PROGRAM A_2_PRG_MachineCtrl
VAR
/////////////////////////////////////////////////////////////////////////////////////TIMERS & TRIGGERS/////////////////////////////////////////////////////////////////////////////////////

	tonSys_Init					: Tc2_Standard.TON:=(PT:=T#1S);
	tonSys_InitTimeout			: Tc2_Standard.TON:=(PT:=T#20S);					
	tonFirstAutoCycle			: Tc2_Standard.TON:=(PT:=T#500MS);
	
/////////////////////////////////////////////////////////////////////////////////////PROCESS CYCLE/////////////////////////////////////////////////////////////////////////////////////	
	
	eCycleState					: E_ProcessCycle;
	tonCMD_Done					: TON;
	tonResetAllCMD				: TON;
	tonExecute					: TON;
	tonSave_Data				: TON;
	tonWriteToCsv				: TON;
	rNoAutoCycle				: R_TRIG;
	
	bStartProcessCondition		: BOOL;
	bIndexDataHistoryFlag		: BOOL;
	rIndexDataHistoryFlag		: R_TRIG;
	bPASS						: BOOL;
	bFAIL						: BOOL;
	i							: INT;
	

	
END_VAR

/////////////////////////////////////////////////////////////////////////////////////GENERAL/////////////////////////////////////////////////////////////////////////////////////
a_ACT_MachineStatus();
b_ACT_ProcessCycle();

ACTION a_ACT_MachineStatus:
/////////////////////////////////////////////////////////////////////////////////////TIMERS/////////////////////////////////////////////////////////////////////////////////////
tonSys_Init(IN:=stMachineStatus.bInitialising);
tonSys_InitTimeout(IN:=stMachineStatus.bInitialising);


/////////////////////////////////////////////////////////////////////////////////////CONDITIONS/////////////////////////////////////////////////////////////////////////////////////
				IF NOT stMasterCtrl.bNoImmediateFault THEN
					stMachineStatus.eMachineState 		:= E_MachineState.IMMEDIATE_FAULT;
				END_IF
				
				IF stMachineStatus.eMachineState		= E_MachineState.STOPPING OR
				stMachineStatus.eMachineState			= E_MachineState.IMMEDIATE_FAULT OR
				stMachineStatus.eMachineState			= E_MachineState.CYCLE_STOP_FAULT THEN
					
					CMD_Station1.bAbort					:= TRUE;	
					CMD_Station2.bAbort					:= TRUE;	
					CMD_Station3.bAbort					:= TRUE;
				
					CMD_Station1.bEnable				:= FALSE;
					CMD_Station2.bEnable				:= FALSE;
					CMD_Station3.bEnable				:= FALSE;
					
				END_IF
				
				IF 	stButtonsLamps.bResetButtonFallingEdge THEN
					CMD_Station1.bReset					:= TRUE;
					CMD_Station2.bReset					:= TRUE;
					CMD_Station3.bReset					:= TRUE;
				ELSE 
					CMD_Station1.bReset					:= FALSE;
					CMD_Station2.bReset					:= FALSE;
					CMD_Station3.bReset					:= FALSE;
				END_IF		
				
/////////////////////////////////////////////////////////////////////////////////////MACHINE CONTROL/////////////////////////////////////////////////////////////////////////////////////

CASE stMachineStatus.eMachineState OF

E_MachineState.SYSTEM_POWER_UP: 		

				IF tonSystemPowerUP.Q THEN
						stMachineStatus.eMachineState 	:= E_MachineState.IMMEDIATE_STOPPED;//
				END_IF
	
E_MachineState.IMMEDIATE_STOPPED:		

				IF stButtonsLamps.bResetButtonFallingEdge THEN
						stMachineStatus.eMachineState 	:= E_MachineState.SYSTEM_INITIALISING;//
				END_IF	


E_MachineState.SYSTEM_INITIALISING:		
				
				CMD_Station1.bAbort						:= FALSE;	
				CMD_Station2.bAbort						:= FALSE;	
				CMD_Station3.bAbort						:= FALSE;	

				IF tonSys_Init.Q THEN
					CMD_Station1.bEnable				:= TRUE;
					CMD_Station2.bEnable				:= TRUE;
					CMD_Station3.bEnable				:= TRUE;						
				END_IF

				IF B_1_1_PRG_Master_Station_1.STATUS.bReady AND B_2_1_PRG_Master_Station_2.STATUS.bReady AND B_3_1_PRG_Master_Station_3.STATUS.bReady THEN 
					stMachineStatus.eMachineState		:= E_MachineState.SYSTEM_READY_TO_START;
				ELSIF stButtonsLamps.bStopButtonFallingEdge OR  
				stMasterCtrl.bCycleStopRequest OR tonSys_InitTimeout.Q THEN
					stMachineStatus.eMachineState 		:= E_MachineState.STOPPING;	
				ELSIF NOT stMasterCtrl.bNoCycleStopFault THEN		
					stMachineStatus.eMachineState 		:= E_MachineState.CYCLE_STOP_FAULT;
				END_IF
			
					
E_MachineState.SYSTEM_READY_TO_START:	

				IF 	 stButtonsLamps.bStartButtonFallingEdge AND stMasterCtrl.bAllStationsReady THEN
					stMachineStatus.eMachineState 		:= E_MachineState.SYSTEM_AUTO_CYCLE;
				ELSIF stButtonsLamps.bStopButtonFallingEdge THEN
					stMachineStatus.eMachineState 		:= E_MachineState.STOPPING;		
				ELSIF stMasterCtrl.bNoCycleStopFault THEN	
					stMachineStatus.eMachineState 		:= E_MachineState.CYCLE_STOP_FAULT;
				ELSIF GVL_Master.stMasterCTRL.bManualModeRequest AND stMasterCtrl.bNoCycleStopFault THEN
					stMachineStatus.eMachineState 		:= E_MachineState.MANUAL_MODE;
				END_IF

				

E_MachineState.SYSTEM_AUTO_CYCLE:		

				IF stButtonsLamps.bStopButtonFallingEdge OR stMasterCtrl.bCycleStopRequest THEN					
					stMachineStatus.eMachineState 		:= E_MachineState.STOPPING;
				ELSIF NOT stMasterCtrl.bNoCycleStopFault THEN	
					stMachineStatus.eMachineState 		:= E_MachineState.CYCLE_STOP_FAULT;
				END_IF
				
E_MachineState.SYSTEM_STANDBY:



E_MachineState.STOPPING:	

				IF stMasterCtrl.bAllStationsStopped THEN
					stMachineStatus.eMachineState 		:= E_MachineState.CYCLE_STOPPED;
				ELSIF NOT stMasterCtrl.bNoCycleStopFault THEN	
					stMachineStatus.eMachineState 		:= E_MachineState.CYCLE_STOP_FAULT;					
				END_IF

E_MachineState.CYCLE_STOPPED:			

				IF stMasterCtrl.bNoCycleStopFault   AND NOT stMasterCtrl.bCycleStopRequest  AND stButtonsLamps.bResetButtonFallingEdge THEN	
					stMachineStatus.eMachineState 		:= E_MachineState.SYSTEM_INITIALISING;		
				END_IF	

E_MachineState.IMMEDIATE_FAULT:	
				
				IF stMasterCtrl.bNoImmediateFault	THEN
					stMachineStatus.eMachineState		:= E_MachineState.IMMEDIATE_STOPPED;		
				END_IF

E_MachineState.CYCLE_STOP_FAULT:		
				
				IF stMasterCtrl.bNoCycleStopFault AND stMasterCtrl.bAllStationsStopped THEN
					stMachineStatus.eMachineState 		:= E_MachineState.CYCLE_STOPPED;
				END_IF	


E_MachineState.MANUAL_MODE:

				IF stButtonsLamps.bStopButtonFallingEdge OR NOT GVL_Master.stMasterCTRL.bManualModeRequest THEN
					stMachineStatus.eMachineState 		:= E_MachineState.STOPPING;
				ELSIF  NOT stMasterCtrl.bNoCycleStopFault THEN	
					stMachineStatus.eMachineState 		:= E_MachineState.CYCLE_STOP_FAULT;								
				ELSE 
					CMD_Station1.bManualMode			:=TRUE;
					CMD_Station2.bManualMode			:=TRUE;
					CMD_Station3.bManualMode			:=TRUE;
				END_IF
ELSE
stMachineStatus.eMachineState:=E_MachineState.SYSTEM_POWER_UP;		
END_CASE									


/////////////////////////////////////////////////////////////////////////////////////MACHINE STATUS/////////////////////////////////////////////////////////////////////////////////////
stMachineStatus.bSystemPowerUp 			:= (stMachineStatus.eMachineState = E_MachineState.SYSTEM_POWER_UP);
stMachineStatus.bImmediateStopped 		:= (stMachineStatus.eMachineState = E_MachineState.IMMEDIATE_STOPPED);
stMachineStatus.bInitialising 			:= (stMachineStatus.eMachineState = E_MachineState.SYSTEM_INITIALISING);
stMachineStatus.bReadyToStart 			:= (stMachineStatus.eMachineState = E_MachineState.SYSTEM_READY_TO_START);
stMachineStatus.bAutoCycle 				:= (stMachineStatus.eMachineState = E_MachineState.SYSTEM_AUTO_CYCLE);
stMachineStatus.bStandby 				:= (stMachineStatus.eMachineState = E_MachineState.SYSTEM_STANDBY);
stMachineStatus.bStopping 				:= (stMachineStatus.eMachineState = E_MachineState.STOPPING);
stMachineStatus.bCycleStopped 			:= (stMachineStatus.eMachineState = E_MachineState.CYCLE_STOPPED);
stMachineStatus.bImmediateFault 		:= (stMachineStatus.eMachineState = E_MachineState.IMMEDIATE_FAULT);
stMachineStatus.bCycleStopFault 		:= (stMachineStatus.eMachineState = E_MachineState.CYCLE_STOP_FAULT);
stMachineStatus.bManualMode 			:= (stMachineStatus.eMachineState = E_MachineState.MANUAL_MODE);

/////////////////////////////////////////////////////////////////////////////////////FLAGS/////////////////////////////////////////////////////////////////////////////////////
stMasterCtrl.bAllStationsStopped		:= (B_1_1_PRG_Master_Station_1.STATUS.bReady AND B_2_1_PRG_Master_Station_2.STATUS.bReady AND B_3_1_PRG_Master_Station_3.STATUS.bReady ) OR
										   (NOT B_1_1_PRG_Master_Station_1.STATUS.bBusy AND NOT B_2_1_PRG_Master_Station_2.STATUS.bBusy AND NOT B_3_1_PRG_Master_Station_3.STATUS.bBusy );
										   
stMasterCtrl.bAllStationsReady			:= B_1_1_PRG_Master_Station_1.bReady AND B_2_1_PRG_Master_Station_2.bReady AND B_3_1_PRG_Master_Station_3.bReady;
END_ACTION

ACTION b_ACT_ProcessCycle:
/////////////////////////////////////////////////////////////////////////////////////UTILITIES & TRIGGERS/////////////////////////////////////////////////////////////////////////////////////

tonCMD_Done( IN := , PT := T#500MS);
tonSave_Data( IN :=  eCycleState = E_ProcessCycle.SAVE_DATA2, PT := T#500MS);
tonResetAllCMD( IN := eCycleState = E_ProcessCycle.RESET_ALL_CMD, PT := T#500MS);
tonWriteToCsv( IN := eCycleState = E_ProcessCycle.CSV, PT := T#500MS);

tonExecute( IN := 	eCycleState = E_ProcessCycle.STATION1_MOV1 OR
					eCycleState = E_ProcessCycle.STATION2_MOV2 OR
					eCycleState = E_ProcessCycle.STATION1_MOV3_STATION2_MOV2 OR
					eCycleState = E_ProcessCycle.STATION3_MOV3,
					PT := T#500MS);
				

rNoAutoCycle( CLK := stMachineStatus.bAutoCycle);

/////////////////////////////////////////////////////////////////////////////////////CONDITIONS/////////////////////////////////////////////////////////////////////////////////////

//bStartProcessCondition := ; //

IF rNoAutoCycle.Q THEN
	eCycleState												:= E_ProcessCycle.RESET_ALL_CMD;
END_IF


CASE eCycleState OF
	
E_ProcessCycle.RESET_ALL_CMD:

				stStation1.Mov1								:= FALSE;
				stStation1.Mov2								:= FALSE;
				stStation1.Mov3								:= FALSE;
				B_1_1_PRG_Master_Station_1.CMD.bExecute		:= FALSE;
				B_1_1_PRG_Master_Station_1.CMD.bReady 		:= FALSE;
				stStation2.Mov1								:= FALSE;
				stStation2.Mov2								:= FALSE;
				stStation2.Mov3								:= FALSE;
				B_2_1_PRG_Master_Station_2.CMD.bExecute		:= FALSE;
				B_2_1_PRG_Master_Station_2.CMD.bReady 		:= FALSE;
				stStation3.Mov1								:= FALSE;
				stStation3.Mov2								:= FALSE;
				stStation3.Mov3								:= FALSE;
				B_3_1_PRG_Master_Station_3.CMD.bExecute		:= FALSE;
				B_3_1_PRG_Master_Station_3.CMD.bReady 		:= FALSE;
				stCSVProcess.bWriteData						:= FALSE;
				
				//bIndexDataHistoryFlag						:= FALSE;
				
				
				IF tonResetAllCMD.Q AND stMachineStatus.bAutoCycle THEN
					eCycleState								:= E_ProcessCycle.IDLE;						
				END_IF
	
E_ProcessCycle.IDLE:
				
				IF bStartProcessCondition AND B_1_1_PRG_Master_Station_1.STATUS.bReady THEN
					eCycleState								:= E_ProcessCycle.STATION1_MOV1;
				END_IF
							
E_ProcessCycle.STATION1_MOV1:

				stStation1.Mov1								:= TRUE;
				B_1_1_PRG_Master_Station_1.CMD.bExecute		:= TRUE;
				
				IF tonExecute.Q THEN
					eCycleState								:= E_ProcessCycle.WAIT_STATION1_MOV1;	
				END_IF

E_ProcessCycle.WAIT_STATION1_MOV1:
				
				IF B_1_1_PRG_Master_Station_1.STATUS.bDone THEN
					eCycleState								:= E_ProcessCycle.STATION2_MOV2;
					stStation1.Mov1							:= FALSE;
					B_1_1_PRG_Master_Station_1.CMD.bExecute	:= FALSE;
					B_1_1_PRG_Master_Station_1.CMD.bReady 	:= TRUE;
				END_IF

E_ProcessCycle.STATION2_MOV2:

				B_1_1_PRG_Master_Station_1.CMD.bReady 		:= FALSE;
				
				stStation2.Mov2								:= TRUE;
				B_2_1_PRG_Master_Station_2.CMD.bExecute		:= TRUE;
				
				IF tonExecute.Q THEN
					eCycleState								:= E_ProcessCycle.WAIT_STATION2_MOV2;	
				END_IF

E_ProcessCycle.WAIT_STATION2_MOV2:

				IF B_2_1_PRG_Master_Station_2.STATUS.bDone THEN
					stStation2.Mov2							:= FALSE;
					B_2_1_PRG_Master_Station_2.CMD.bExecute	:= FALSE;
					B_2_1_PRG_Master_Station_2.CMD.bReady 	:= TRUE;	
					eCycleState								:= E_ProcessCycle.STATION1_MOV3_STATION2_MOV2;
				END_IF

E_ProcessCycle.STATION1_MOV3_STATION2_MOV2:

				B_2_1_PRG_Master_Station_2.CMD.bReady 		:= FALSE;
	
				stStation1.Mov3								:= TRUE;
				stStation2.Mov2								:= TRUE;
				B_2_1_PRG_Master_Station_2.CMD.bExecute		:= TRUE;
				B_1_1_PRG_Master_Station_1.CMD.bExecute		:= TRUE;
				
				IF tonExecute.Q THEN
					eCycleState								:= E_ProcessCycle.WAIT_STATION1_MOV3_STATION2_MOV2;	
				END_IF

E_ProcessCycle.WAIT_STATION1_MOV3_STATION2_MOV2:
			
				IF B_2_1_PRG_Master_Station_2.STATUS.bDone AND B_1_1_PRG_Master_Station_1.STATUS.bDone THEN
					stStation1.Mov3							:= FALSE;
					stStation2.Mov2							:= FALSE;
					B_2_1_PRG_Master_Station_2.CMD.bExecute	:= FALSE;
					B_1_1_PRG_Master_Station_1.CMD.bExecute	:= FALSE;	
					B_2_1_PRG_Master_Station_2.CMD.bReady 	:= TRUE;
					B_1_1_PRG_Master_Station_1.CMD.bReady 	:= TRUE;
					eCycleState								:= E_ProcessCycle.STATION3_MOV3;
				END_IF	

E_ProcessCycle.STATION3_MOV3:

					B_2_1_PRG_Master_Station_2.CMD.bReady 	:= FALSE;
					B_1_1_PRG_Master_Station_1.CMD.bReady 	:= FALSE;
					
					B_3_1_PRG_Master_Station_3.CMD.bExecute	:= TRUE;
					stStation3.Mov3							:= TRUE;
					
				IF tonExecute.Q THEN
					eCycleState								:= E_ProcessCycle.WAIT_STATION3_MOV3;	
				END_IF

E_ProcessCycle.WAIT_STATION3_MOV3:

				IF B_3_1_PRG_Master_Station_3.STATUS.bDone THEN
					stStation3.Mov3							:= FALSE;
					B_3_1_PRG_Master_Station_3.CMD.bExecute	:= FALSE;
					B_3_1_PRG_Master_Station_3.CMD.bReady 	:= TRUE;	
					bIndexDataHistoryFlag					:= TRUE;
					eCycleState								:= E_ProcessCycle.SAVE_DATA;
				END_IF

E_ProcessCycle.SAVE_DATA:

				FOR i := 199 TO 0 BY -1 DO
					aDataHistory[i+1] 						:= aDataHistory[i];
				END_FOR			
				eCycleState									:= E_ProcessCycle.SAVE_DATA2;
					
E_ProcessCycle.SAVE_DATA2:	
				
				c_ACT_SaveData();
				IF tonSave_Data.Q THEN
					eCycleState								:= E_ProcessCycle.CSV;
				END_IF	
				
				
E_ProcessCycle.CSV:
			
				stCSVProcess.bWriteData						:= TRUE;
				IF tonWriteToCsv.Q THEN
					stCSVProcess.bWriteData					:= FALSE;
				END_IF
				IF NOT stCSVProcess.bBusy AND tonWriteToCsv.Q THEN
					eCycleState								:= E_ProcessCycle.RESET_ALL_CMD;
					nIndexDataHistory						:= nIndexDataHistory +1;
				END_IF
				
END_CASE
END_ACTION

ACTION c_ACT_SaveData:
(*rIndexDataHistoryFlag( CLK := 	bIndexDataHistoryFlag);
	IF rIndexDataHistoryFlag.Q THEN
					nIndexDataHistory						:= nIndexDataHistory + 1;
					bIndexDataHistoryFlag					:= FALSE;
	END_IF*)

				
	//STATION 1
	aDataHistory[0].sSetting1_1	:= stCycleDataStation1.sSetting1;
	aDataHistory[0].nSetting2_1	:= stCycleDataStation1.nSetting2;
	aDataHistory[0].bSetting3_1	:= stCycleDataStation1.bSetting3;
	
	aDataHistory[0].sDATA1_1	:= stCycleDataStation1.sDATA1;
	aDataHistory[0].nDATA2_1	:= stCycleDataStation1.nDATA2;
	aDataHistory[0].bDATA3_1	:= stCycleDataStation1.bDATA3;
	
	aDataHistory[0].bPass_1		:= stCycleDataStation1.bPass;
	aDataHistory[0].bFail_1		:= stCycleDataStation1.bFail;
	
	//STATION 2
	aDataHistory[0].sSetting1_2	:= stCycleDataStation2.sSetting1;
	aDataHistory[0].nSetting2_2	:= stCycleDataStation2.nSetting2;
	aDataHistory[0].bSetting3_2	:= stCycleDataStation2.bSetting3;
	
	aDataHistory[0].sDATA1_2	:= stCycleDataStation2.sDATA1;
	aDataHistory[0].nDATA2_2	:= stCycleDataStation2.nDATA2;
	aDataHistory[0].bDATA3_2	:= stCycleDataStation2.bDATA3;
	
	aDataHistory[0].bPass_2		:= stCycleDataStation2.bPass;
	aDataHistory[0].bFail_2		:= stCycleDataStation2.bFail;
	
	//STATION 3
	aDataHistory[0].sSetting1_3	:= stCycleDataStation3.sSetting1;
	aDataHistory[0].nSetting2_3	:= stCycleDataStation3.nSetting2;
	aDataHistory[0].bSetting3_3	:= stCycleDataStation3.bSetting3;
	
	aDataHistory[0].sDATA1_3	:= stCycleDataStation3.sDATA1;
	aDataHistory[0].nDATA2_3	:= stCycleDataStation3.nDATA2;
	aDataHistory[0].bDATA3_3	:= stCycleDataStation3.bDATA3;
	
	aDataHistory[0].bPass_3		:= stCycleDataStation3.bPass;
	aDataHistory[0].bFail_3		:= stCycleDataStation3.bFail;
 
	
	
	aDataHistory[0].bPass		:= bPASS;
	aDataHistory[0].bFail		:= bFAIL;
	aDataHistory[0].sData		:= sSystemDate;
	aDataHistory[0].sTime		:= sSystemTime;
END_ACTION

END_PROGRAM

(* stored: Version 1.1.0.1, ProductVersion 3.1.4024.13
   POU A_2_PRG_MachineCtrl: Id {fa5999e8-1190-4f6f-b7ba-be790246df67}, SpecialFunc None
   Action a_ACT_MachineStatus: Id {83375328-405c-4671-a979-0a97efed562c}
   Action b_ACT_ProcessCycle: Id {5e92037d-73c3-401d-956e-95e5929b3e1d}
   Action c_ACT_SaveData: Id {5a28b6f2-a56d-4cef-8c15-c08642850884} *)
